TYPE Buffer_Cnv_Inputs_DUT :
STRUCT
	Forward_Sensor:	BOOL;
	Backward_Sensor:	BOOL;
	Shuttle_High:	BOOL;
	VFD_Status:	WORD;
	VFD_Speed_Actual:	INT;
	VFD_ActualCurrent:	INT;
	VFD_ActualTorque:	INT;
END_STRUCT
END_TYPE

(* stored: Version 1.1.0.1
   DUT Buffer_Cnv_Inputs_DUT: Id {ba3cceb8-ed1d-40d5-a91b-0bc258abdd19} *)
